(* PLC project TemplateSPK1xxM01, CODESYS CODESYS V3.5 SP17 Patch 3 *)
(* stored: creationDateTime 2025-06-01T22:10:51.152379, version 3.5.14.30, modificationDateTime 2025-06-01T22:08:43.545814, organization Production association OWEN *)

TYPE YOUR_STRUCT : STRUCT
  ID : INT;
  Name : WSTRING;
  Value : REAL;
  Sub_1 : YOUR_SUB_STRUCT;
  Sub_2 : YOUR_SUB_STRUCT;
END_STRUCT;
END_TYPE

TYPE JS_YOUR_STRUCT : STRUCT
  ID : JSONVAR;
  Name : JSONVAR;
  Value : JSONVAR;
  Sub_1 : JS_YOUR_SUB_STRUCT;
  Sub_2 : JS_YOUR_SUB_STRUCT;
END_STRUCT;
END_TYPE

TYPE JS_YOUR_SUB_STRUCT : STRUCT
  ID : JSONVAR;
  Sub_value : JSONVAR;
  Direction : JSONVAR;
END_STRUCT;
END_TYPE

TYPE YOUR_SUB_STRUCT : STRUCT
  ID : UINT;
  Sub_value : REAL;
  Direction : BOOL;
END_STRUCT;
END_TYPE

{attribute 'contains_implicit_enum'}
FUNCTION_BLOCK JS_TO_VAR
  VAR_INPUT
    xStart : REFERENCE TO BOOL;
    sFileName : STRING(255);  (* Take care of path. *)
    stResult : REFERENCE TO ARRAY [1..32] OF YOUR_STRUCT;  (* Set here the maximum size of array *)
  END_VAR
  VAR CONSTANT
    iArrayMaxSize : INT := 32;  (* Set here the maximum size of array *)
  END_VAR
  VAR_OUTPUT
    xDone : BOOL;
    xBusy : BOOL;
    xError : BOOL;
  END_VAR
  VAR
    myArray : ARRAY[1..iArrayMaxSize] OF JS_YOUR_STRUCT;  (* !!!! NAME HERE SHOULD MATCH TOPMOST JSON OBJ/// Use refactoring to rename *)
    {attribute 'hide'}
    ParseJSON : JSON_TO_STRUCT;  (* === FB-VALS ===// *)
    reader : ReadJSONFile;
    parsedString : STRING(GPL_JSON.MAX_JSON_STRING);
    i : INT;
    {attribute 'implicit_enum_type'}
    STATE : Implicit_Enum__JS_TO_VAR__STATE;
    xStartPrev : BOOL;
  END_VAR

            CASE STATE OF
	
	IDLE:
		IF xStart AND NOT xStartPrev THEN
			reader.xStart:=TRUE;
			xError:=FALSE;
			xBusy:=TRUE;
			xDone:=FALSE;
			ParseJSON.Execute:=FALSE;
			STATE:=READ;
		END_IF
	
	READ:
		reader(sFileName:=sFileName,Result:=parsedString);
		IF reader.xError THEN
			xError:=TRUE;
			ParseJSON.Execute:=FALSE;
			
			STATE:=FINISH;
		ELSIF reader.xDone THEN
				ParseJSON.Execute:=TRUE;
				STATE:=PARSE;
		END_IF	
	
	PARSE:
		ParseJSON(
			JSONString:= ADR(parsedString), 
			JSONStringSize:= SIZEOF(parsedString),
			JSONVars:= ADR(myArray),
			NumberOfVars:= SIZEOF(myArray) / SIZEOF(JSONVAR)
		);
		IF ParseJSON.Error THEN
			ParseJSON.Execute:=FALSE;
			xError:=TRUE;
			STATE:=FINISH;
		ELSIF ParseJSON.Done THEN
			ParseJSON.Execute:=FALSE;
			STATE:=Convert;
		END_IF
	
	CONVERT:
		FOR i:=1 TO iArrayMaxSize DO
			stResult[i]:=CORE_JS_TO_ST(myArray[i]);
		END_FOR;
		STATE:=FINISH;
	
	FINISH:
		xStart:=FALSE;
		xBusy:=FALSE;
		xDone:=TRUE;
END_CASE
xStartPrev:=xStart;
          

METHOD CORE_JS_TO_ST : YOUR_STRUCT
  VAR_INPUT
    JS : JS_YOUR_STRUCT;
  END_VAR
                  CORE_JS_TO_ST.ID:=TO_INT(JS.ID.Number); 
//Dealing with Cyrillic symbols
CORE_JS_TO_ST.Name:=OSU.CP1251_TO_UNICODE(JS.Name.AsString);
CORE_JS_TO_ST.Value:=JS.Value.Number;
CORE_JS_TO_ST.Sub_1:=SUB_JS_TO_ST(JS.Sub_1);
CORE_JS_TO_ST.Sub_2:=SUB_JS_TO_ST(JS.Sub_2);
                
END_METHOD

METHOD SUB_JS_TO_ST : YOUR_SUB_STRUCT
  VAR_INPUT
    JS : JS_YOUR_SUB_STRUCT;
  END_VAR
                  //Removing all non-numbers and converting to integer
SUB_JS_TO_ST.ID:=STRING_TO_UINT(OSCAT.CLEAN(JS.ID.AsString,'0123456789'));
SUB_JS_TO_ST.Sub_value:=JS.Sub_value.Number;
//Making bool out of some text
SUB_JS_TO_ST.Direction:=(OSCAT.FINDB(JS.Direction.AsString,'UP')>0);

                
END_METHOD
END_FUNCTION_BLOCK

PROGRAM TEST
  VAR
    converter : JS_TO_VAR;
    myST : ARRAY[1..32] OF YOUR_STRUCT;
    xRun : BOOL;
    sFileName : STRING(255) := 'test.json';  (* Default path for virtual controller is C:\ProgramData\CODESYS\CODESYSControlWinV3\FA001425\PlcLogic// Controller version FA001425 may vary. *)
  END_VAR

            converter.sFileName:=sFileName;
converter(stResult:=myST,xStart:=xRun);
          
END_PROGRAM

{attribute 'contains_implicit_enum'}
FUNCTION_BLOCK ReadJSONFile
  VAR CONSTANT
    SplitSize : INT := 2048;
  END_VAR
  VAR_INPUT
    xStart : BOOL;
    sFileName : REFERENCE TO STRING(255);
    Result : REFERENCE TO STRING(GPL_JSON.MAX_JSON_STRING);
  END_VAR
  VAR_OUTPUT
    xBusy : BOOL;
    xDone : BOOL;
    xError : BOOL;
  END_VAR
  VAR
    fopen : FILE.Open;
    fread : FILE.Read;
    fclose : FILE.Close;
    xStartPrev : BOOL;
    {attribute 'implicit_enum_type'}
    step : Implicit_Enum__ReadJSONFile__step;
    tempString : STRING(GPL_JSON.MAX_JSON_STRING);
    endPos : INT;
    subString : STRING(SplitSize);  (* Not more than CLEANSTRING.MAXSTRING; *)
    cleanupCount : INT := 0;
    cleanupCounter : INT;
    tmp : REAL;
    start : INT;
    finish : INT;
    lenCopy : INT;
  END_VAR

            CASE step OF
	IDLE:
		IF xStart AND NOT xStartPrev THEN
			step:=OPEN;
			xDone:=FALSE;
			xBusy:=TRUE;
			xError:=FALSE;
			
		END_IF
		
		fopen(xExecute:=FALSE);
    	fread(xExecute:=FALSE);
		fclose(xExecute:=FALSE);
	
	OPEN:
		fopen.sFileName:=sFileName;
		fopen.eFileMode:=FILE.MODE.MREAD;
		fopen.xExclusive:=TRUE;
		fopen(xExecute:=TRUE);
		
		IF fopen.xDone THEN
			step:=READ;
		END_IF
		IF fopen.xError THEN
			step:=CLOSE;
			xError:=TRUE;
		END_IF
		
	READ:
		Result:='';
		fread.hFile:=fopen.hFile;
		
		fread.pBuffer:=ADR(tempString);
		
		fread.szBuffer:=SIZEOF(tempString);
		fread(xExecute:=TRUE);
		IF fread.xDone THEN
			step:=CLEANUP;
			endPos:=TO_INT(StrLenA(ADR(tempString)));
			start:=1;
			cleanupCounter:=0;
			
			cleanupCount:=TO_INT(endPos/SplitSize);
			//Simple Round up
			tmp:=TO_REAL(endPos)/TO_REAL(SplitSize);
			IF tmp>TO_REAL(cleanupCount) THEN
				cleanupCount:=cleanupCount+1;
			END_IF
			
		END_IF
		IF fread.xError THEN
			step:=CLOSE;
			xError:=TRUE;
		END_IF
	CLEANUP:
		
		finish:=MIN(endPos,start+SplitSize);
		
		lenCopy:=MIN(SplitSize,endPos-start+1);
		IF lenCopy>0 THEN
		
			STU.StrMidA(ADR(tempString),SIZEOF(tempString),lenCopy,start,ADR(subString),SplitSize);
			CLEANSTRING(ADR(subString));
			STU.StrConcatA(ADR(subString),ADR(Result),SIZEOF(Result));
		END_IF
		
		IF finish>=endPos THEN //Somewhow this does not work even then true...
			step:=CLOSE;
		END_IF
		
		start:=start+SplitSize;
		cleanupCounter:=cleanupCounter+1;
		IF cleanupCounter>cleanupCount THEN //So double-check it.
			step:=CLOSE;
		END_IF
	CLOSE:
		fclose.hFile:=fopen.hFile;
		fclose(xExecute:=TRUE);
		IF fclose.xDone THEN
			step:=FINISH;
		END_IF
		IF fclose.xError THEN
			step:=FINISH;
			xError:=TRUE;
		END_IF
		
	FINISH:
		step:=IDLE;
		xDone:=TRUE;
		xStart:=FALSE;
		xBusy:=FALSE;
END_CASE
xStartPrev := xStart;
          
END_FUNCTION_BLOCK
